	//=============================================================================
	// EXISTING DEVICES
	//=============================================================================
	#tempRetValDeviceStates := DeviceStates(LADDR := #ioSystemHwId,
	                                        MODE := #STATE_EXIST,
	                                        STATE := #statExistingDevices);

	// Check if the block call was successful
	IF (#tempRetValDeviceStates <> 0)
	THEN
	    // Error handling
	    #status := #tempRetValDeviceStates;
	    #instructionError := #ERR_DEV_STATE_DEVICES;
	    // Call ok --> store the actual number of configured devices
	ELSE
	    ;
	END_IF;

	//=============================================================================
	// FAULTY DEVICES
	//=============================================================================
	#tempRetValDeviceStates := DeviceStates(LADDR := #ioSystemHwId,
	                                        MODE := #STATE_FAULTY,
	                                        STATE := #statFaultyDevices);

	// Check if the block call was successful
	IF (#tempRetValDeviceStates <> 0)
	THEN
	    // Error handling
	    #status := #tempRetValDeviceStates;
	    #instructionError := #ERR_DEV_STATE_DEVICES;
	    // Call ok --> store the actual number of configured devices
	ELSE
	    ;
	END_IF;

	// Find out the number of the assigned IO system, to define if it is
	// a PN or DP Network
	#tempRetValGeo := LOG2GEO(LADDR := #ioSystemHwId,
	                          GEOADDR := #statGeoAddr);

	// set IO system ID
	#ioSystem.ioSystemId := #statGeoAddr.IOSYSTEM;

	// Inilize the structure for system function GEO2LOG
	#statGeoAddr.HWTYPE := #DEVICE_SLAVE;   // Hardware type 2: IO device
	// Predefine the type OF IO system. Either Profinet IO or Profibus DP
	IF ((#statGeoAddr.IOSYSTEM >= 100)
	    AND (#statGeoAddr.IOSYSTEM <= 115))
	THEN
	    #statGeoAddr.AREA := #IO_SYSTEM_AREA;   // Area ID 1: PROFINET IO
	    #statMaxDevices := #MAX_SLAVES_PN;
	ELSIF ((#statGeoAddr.IOSYSTEM >= 1)
	    AND (#statGeoAddr.IOSYSTEM <= 32))
	THEN
	    #statGeoAddr.AREA := #DP_SYSTEM_AREA;   // Area ID 1: Profibus DP
	    #statMaxDevices := #MAX_SLAVES_DP;
	ELSE
	    ;
	END_IF;

	// Go trough all devices and get the status of the configured
	FOR #tempIndex := 1 TO #statMaxDevices DO
	    // The devices are configured --> Read out the logical address and the
	    // device name
	    IF (#statConfiguredDevices[#tempIndex] = TRUE)
	    THEN
	        // Increment the actual configured devices, store the state and
	        // HW_ID as an numerical value (UINT)
	        #statActualConfiguredDevices := #statActualConfiguredDevices + 1;

	        // Store the first configured device for the linked list
	        IF (#statFirstDeviceFlag = TRUE)
	        THEN
	            #statFirstDevice := INT_TO_UINT(#tempIndex);
	            #ioSystem.firstDevice := UINT_TO_INT(#statFirstDevice);
	            #statFirstDeviceFlag := FALSE;
	            #tempLastDevice := INT_TO_UINT(#tempIndex);
	            // It is not the first bit --> Store the actual index as "next device"
	            // in the further one!
	        ELSE
	            #ioSystem.device[#tempLastDevice].nextDevice := #tempIndex;
	            #tempLastDevice := INT_TO_UINT(#tempIndex);
	        END_IF;
	        // Store the index of the last device for the exit condition of the
	        // followiing instructions
	        #statLastDevice := #tempLastDevice;
	        #ioSystem.lastDevice := UINT_TO_INT(#statLastDevice);

	        // Station number
	        #statGeoAddr.STATION := INT_TO_UINT(#tempIndex);
	        // read LADDR from devices
	        #tempRetValGeo := GEO2LOG(GEOADDR := #statGeoAddr,
	                                  LADDR => #statGeoLaddr);
	        // Everything is ok!
	        IF (#tempRetValGeo = 0)
	        THEN
	            // store LADDR from devices in diagnostic data block
	            #ioSystem.device[#tempIndex].laddr := #statGeoLaddr;

	            // Store the device name, if the device is existing
	            // Get name is an acyclic instruction. In the startup OB, the
	            // instruction has to be repeated until it is done or error
	            REPEAT
	                // Get device name of each decive in PN System
	                #instGetNameDevices(LADDR := #ioSystemHwId,
	                                    STATION_NR := #statGeoAddr.STATION,
	                                    DATA := #tempStringConvert);

	            UNTIL (#instGetNameDevices.DONE = TRUE)
	                OR (#instGetNameDevices.ERROR = TRUE)
	            END_REPEAT;

	            IF (#instGetNameDevices.ERROR = TRUE)
	            THEN
	                // Error handling
	                #status := WORD_TO_INT(#instGetNameDevices.STATUS);
	                #instructionError := #ERR_GET_NAME_DEVICES;
	                #errorIndex := #tempIndex;

	                // Everything is ok --> Convert the String[254] into String[50]
	            ELSIF (#instGetNameDevices.DONE = TRUE)
	            THEN
	                // Cut all characters more than 50 to reduce the string length
	                #ioSystem.device[#tempIndex].name := DELETE(IN := #tempStringConvert,
	                                                            L := 204,
	                                                            P := 50);

	                // Initialize the temporary string before next loop
	                #tempStringConvert := #statInitString;
	            ELSE
	                ;
	            END_IF;
	        ELSE
	            // If the return value ist not = 0 --> the device/system/module is
	            // not configured --> No error handling
	            // set LADDR from devices to 0 in diagnostic data block
	            #ioSystem.device[#tempIndex].laddr := 0;
	            #ioSystem.device[#tempIndex].name := '';
	        END_IF;

	        // Check if the configured devices are faulty or lost once through
	        // the startup!
	        IF (#statExistingDevices[#tempIndex] = TRUE)
	        THEN
	            IF (#statFaultyDevices[#tempIndex] = TRUE)
	            THEN

	                #ioSystem.device[#tempIndex].errorState := 2;
	                #ioSystem.device[#tempIndex].error := TRUE;

	                // The device is not faulty and does exist --> set state ok!
	            ELSE
	                #ioSystem.device[#tempIndex].errorState := 1;
	                #ioSystem.device[#tempIndex].error := FALSE;
	            END_IF;
	            // The connection to the device is lost at the moment
	        ELSE
	            #ioSystem.device[#tempIndex].errorState := 3;
	            #ioSystem.device[#tempIndex].error := TRUE;
	        END_IF;
	        // No device is configured
	    ELSE
	        ;
	    END_IF;

	END_FOR;
	// Store the actual configured devices in the diagnostics structure
	#ioSystem.actualConfiguredDevices := #statActualConfiguredDevices;

	// Mark parameter "Next Device" of the last device in the list
	// --> "Next Device" = negative --> Last device in the list
	#ioSystem.device[#statLastDevice].nextDevice := -1;

	// Go through the devices until the last device is reached
	// If there are gaps between the device-list, jump over and have a look on
	// the "NextDevice" parameter
	REPEAT
	    IF (#statFirstRun = TRUE)
	    THEN
	        // The index of the linked list is representing the station number.
	        #statGeoAddr.STATION := #statFirstDevice;
	        // Initialize the pointer for the first run
	        #statLinkedListPointer := UINT_TO_INT(#statFirstDevice);
	        // Reset the flag, which signalizes the first run.
	        #statFirstRun := FALSE;
	    ELSE
	        // The index of the linked list is representing the station number.
	        #statGeoAddr.STATION := INT_TO_UINT(#statLinkedListPointer);
	    END_IF;

	    //=============================================================================
	    // Get the logical address of all modules and store the actual number of
	    // modules from each device
	    //=============================================================================

	    // Inilize the structure for system function GEO2LOG
	    #statGeoAddr.HWTYPE := #MODULE_OF_DEVICE;   // Hardware type 4: Module
	    FOR #tempModuleNum := 0 TO 10 DO
	        // Slot number
	        #statGeoAddr.SLOT := INT_TO_UINT(#tempModuleNum);
	        // read LADDR from modules
	        #tempRetValGeo := GEO2LOG(GEOADDR := #statGeoAddr,
	                                  LADDR => #statGeoLaddr);
	        // check Retval
	        IF (#tempRetValGeo = 0)
	        THEN
	            // store LADDR from modules in diagnostic data block
	            #ioSystem.device[#statLinkedListPointer].slot[#tempModuleNum].slotLaddr := #statGeoLaddr;
	            #ioSystem.device[#statLinkedListPointer].actualConfiguredModules := #ioSystem.device[#statLinkedListPointer].actualConfiguredModules + 1;
	        ELSE
	            // If the return value ist not = 0 --> the device/system/module is
	            // not configured --> No error handling
	            // set LADDR from modules to 0 in diagnostic data block
	            #ioSystem.device[#statLinkedListPointer].slot[#tempModuleNum].slotLaddr := 0;
	        END_IF;
	    END_FOR;

	    //=============================================================================
	    // Check modules of faulty Devices
	    //=============================================================================

	    // Check the state of the configured devices
	    IF (#ioSystem.device[#statLinkedListPointer].errorState = 2)
	    THEN
	        // The device is reachable, but faulty because of an error in a
	        // subordinated system --> check the modules
	        #tempRetValModuleStates := ModuleStates(LADDR := #ioSystem.device[#statLinkedListPointer].laddr,
	                                                MODE := #STATE_PROBLEM,
	                                                STATE := #statDeviceModuleStates);

	        IF (#tempRetValModuleStates <> 0)
	        THEN
	            // Error hanlding
	            #status := #tempRetValModuleStates;
	            #instructionError := #ERR_MOD_STAT_DEVICES;
	            #errorIndex := UINT_TO_INT(#statFirstDevice);
	        ELSE
	            // Store the state of the different module in the diag DB
	            FOR #tempSlotIndex := 0 TO #ioSystem.device[#statFirstDevice].actualConfiguredModules DO
	                IF (#statDeviceModuleStates[#tempSlotIndex + 1] = TRUE)
	                THEN
	                    #ioSystem.device[#statLinkedListPointer].slot[#tempSlotIndex].slotErrorState := TRUE;
	                ELSE
	                    #ioSystem.device[#statLinkedListPointer].slot[#tempSlotIndex].slotErrorState := FALSE;
	                END_IF;
	            END_FOR;
	        END_IF;
	    ELSIF (#ioSystem.device[#statLinkedListPointer].errorState = 3)
	    THEN

	        FOR #tempSlotIndex := 0 TO #ioSystem.device[#statLinkedListPointer].actualConfiguredModules DO
	            IF (#ioSystem.device[#statLinkedListPointer].slot[#tempSlotIndex].slotLaddr <> 0)
	            THEN
	                #ioSystem.device[#statLinkedListPointer].slot[#tempSlotIndex].slotErrorState := TRUE;
	            END_IF;
	        END_FOR;

	    ELSE
	        ; // no faulty device --> nothing to do!
	    END_IF;

	    // Initialize the pointer for the next run
	    #statLinkedListPointer := #ioSystem.device[#statLinkedListPointer].nextDevice;
	    // If the last device is reached, reset the bit for the first run
	    //#FirstRun := TRUE;
	    // Checking the modules is done, the last device is reached
	UNTIL (#statLinkedListPointer < 0)
	END_REPEAT;
	// Reset the condition for the first run.
	#statFirstRun := TRUE;


END_FUNCTION_BLOCK

DATA_BLOCK "DiagStartupIoSystem_iDB"
{ S7_Optimized_Access := 'TRUE' }
VERSION : 0.1
NON_RETAIN
"DiagStartupIoSystem"

BEGIN

END_DATA_BLOCK

FUNCTION_BLOCK "DiagStartupPlc"
{ S7_Optimized_Access := 'TRUE' }
VERSION : 0.1
   VAR_OUTPUT
      status : Int;   // The return value of system function, where the last error occured
      instructionError : Int;   // Indicates in which system function the error occured: 1= DeviceStates PN , 2=GetName PN, 3=ModuleStates PN,  4=DeviceStates DP, 5= GetName DP. 6= ModuleStates DP
   END_VAR

   VAR_IN_OUT
      plc : "typePlc";   // The diagnostics structure for one PLC
   END_VAR

   VAR
      statGeoAddr {OriginalPartName := 'GEOADDR'; LibVersion := '1.0'; ExternalAccessible := 'False'; ExternalVisible := 'False'; ExternalWritable := 'False'} : GEOADDR;   // Slot information
      statGeoLaddr { ExternalAccessible := 'False'; ExternalVisible := 'False'; ExternalWritable := 'False'} : HW_ANY;   // GEO2LOG hardware identifier
      statActualCentralModules : USInt := 0;   // Actual number of modules in the central station (PLC)
      statPlcModuleStates : Array[0..127] of Bool;   // Storage of the status of all modules in the PLC central station --> State: Problem
   END_VAR

   VAR_TEMP
      tempModuleNum : Int;   // index module number
      tempRetValGeo : Int;   // GEO2LOG error information
      tempRetValModuleStates : Int;   // Return value system function ModuleStates
   END_VAR

   VAR CONSTANT
      MODULE_OF_PLC : USInt := 4;   // GEO2LOG structure: HW type = 4
      CPU : USInt := 0;   // GEO2LOG structure: Area = 0
      CENTRAL_SYSTEM : USInt := 0;   // GEO2LOG structure: IO System = 0
      CENTRAL_STATION : USInt;   // GEO2LOG structure: Station = 0
      HW_ID_PLC_MODULES : HW_DEVICE := 32;   // HW ID of the PLC, which is needed for getting the module states --> fix value
      STATE_PROBLEM : USInt := 5;   // Used for instruction DeviceStates, read out all devices with several problems
      ERR_MOD_STAT_CENTRAL : USInt := 3;   // Value for output instruction error, ModuleStates local modules
   END_VAR


BEGIN
	//=============================================================================
	//Author: SIEMENS, Owner: Miklos Boros
	//        email: borosmiklos@gmail.com; miklos.boros@esss.se
	//
	//Functionality: Determine hardware identifier and module states from local
	//               modules
	//
	//
	//Please Note:
	//        This block is part of the generated ESS Standard Code
	//        DON'T CHANGE THIS BLOCK MANUALY. Any changes will be overwritten in the next code generation.
	//
	//
	//Change log table:
	//Version  Date         Expert in charge      Changes applied
	//01.00.00 29.08.2017   ESS/ICS               First released version for PLCFactory
	//02.00.00 09-04-2018   ESS/ICS               Major bug fix for PN/DP devices
	//=============================================================================


	//=============================================================================
	// Determine hardware identifier from LOCAL MODULES
	//=============================================================================
	#statGeoAddr.HWTYPE := #MODULE_OF_PLC;      // Hardware type 4: module
	#statGeoAddr.AREA := #CPU;                  // Area ID 0: CPU
	#statGeoAddr.IOSYSTEM := #CENTRAL_SYSTEM;   // PROFINET IO system
	                                            // (0 = central unit in the rack)
	#statGeoAddr.STATION := #CENTRAL_STATION;   // Number of the rack
	                                            // if area identifier
	                                            //  AREA = 0 (central module).

	FOR #tempModuleNum := 1 TO 10 DO
	  // Slot number
	  #statGeoAddr.SLOT := INT_TO_UINT(#tempModuleNum);
	  // read LADDR from local modules
	  #tempRetValGeo := GEO2LOG(GEOADDR := #statGeoAddr,
	                            LADDR => #statGeoLaddr);
	  // check Retval
	  IF (#tempRetValGeo = 0)
	  THEN
	    // store LADDR from local modules in diagnostic data block
	    #plc.slot[#tempModuleNum].slotLaddr := #statGeoLaddr;
	    #statActualCentralModules := #statActualCentralModules + 1;
	  ELSE
	    // If the return value ist not = 0 --> the device/system/module is not
	    // configured --> No error handling
	    // set LADDR from local modules to 0 in diagnostic data block
	    #plc.slot[#tempModuleNum].slotLaddr := 0;
	  END_IF;
	  // Store the actual configured devices in the diagnostics DB
	  #plc.actualConfiguredCentralModules := #statActualCentralModules;
	END_FOR;


	//=============================================================================
	// Check module states from LOCAL MODULES
	//=============================================================================
	// Check if central module are available - at least one module is always
	// configured, the PLC itself
	IF (#plc.actualConfiguredCentralModules > 1)
	THEN
	  // Check the status of the local modules
	  #tempRetValModuleStates := ModuleStates(LADDR := #HW_ID_PLC_MODULES,
	                                          MODE := #STATE_PROBLEM,
	                                          STATE := #statPlcModuleStates);

	  // Check if the block call was successful
	  IF (#tempRetValModuleStates <> 0)
	  THEN
	    // Error handling
	    #status := #tempRetValModuleStates;
	    #instructionError := #ERR_MOD_STAT_CENTRAL;
	  ELSE
	    ; // Everything is ok!
	  END_IF;
	ELSE
	  ; // There are no central module configured
	END_IF;

	// The error LED of the PLC is flashing --> Set error state of the PLC
	#plc.errorState := TRUE;


	//=============================================================================
	// set module states from LOCAL MODULES
	//=============================================================================

	// If the first bit in the array is true, at least one module is faulty
	IF (#statPlcModuleStates[0] = TRUE)
	THEN
	  // Check which of the modules are faulty
	  // PLC modules array starts at index 2 for the first local module
	  FOR #tempModuleNum := 2 TO #plc.actualConfiguredCentralModules + 1 DO
	    IF (#statPlcModuleStates[#tempModuleNum] = TRUE)
	    THEN
	      #plc.slot[#tempModuleNum - 1].slotErrorState := TRUE;
	    ELSE
	      #plc.slot[#tempModuleNum - 1].slotErrorState := FALSE;
	    END_IF;
	  END_FOR;

	ELSE
	  // Everything is ok!
	  FOR #tempModuleNum := 1 TO #plc.actualConfiguredCentralModules DO
	    #plc.slot[#tempModuleNum].slotErrorState := FALSE;
	  END_FOR;

	END_IF;

END_FUNCTION_BLOCK


DATA_BLOCK "DiagStartupPlc_iDB"
{ S7_Optimized_Access := 'TRUE' }
VERSION : 0.1
NON_RETAIN
"DiagStartupPlc"

BEGIN

END_DATA_BLOCK

FUNCTION "DiagnosticError" : Void
{ S7_Optimized_Access := 'TRUE' }
VERSION : 0.1
   VAR_INPUT
      ioState : Word;   // IO state of the HW object
      laddr : HW_ANY;   // Hardware identifier
      channel : UInt;   // Channel number
      multiError : Bool;   // =true if more than one error is present
   END_VAR

   VAR_IN_OUT
      plc : "typePlc";   // The diagnostics structure for one PLC
      ioSystem : Array[1..5] of "typeIoSystem";   // The diagnostics structure for one IO System
   END_VAR

   VAR_TEMP
      tempGeoAddr {OriginalPartName := 'GEOADDR'; LibVersion := '1.0'} : GEOADDR;   // Geographical address of the disturbed Module / Device
      tempIoSystemIndex : Int;   // Index for IO System
      index : Int;   // index system
      tempRetVal : Int;   // Return value of LOG2GEO
   END_VAR

   VAR CONSTANT
      GOOD : Word := 16#0001;   // Status of the hardware object: Bit 0: Good
      AREA_CENTRAL : UInt := 0;   // Area ID for PLC
      AREA_PROFINET : UInt := 1;   // Area ID for PROFINET IO
      AREA_PROFIBUS : UInt := 2;   // Area ID for PROFIBUS DP
   END_VAR


BEGIN
	//=============================================================================
	//Author: SIEMENS, Owner: Miklos Boros
	//        email: borosmiklos@gmail.com; miklos.boros@esss.se
	//
	//Functionality: Evaluate Diagnostic interrupt OB information for PLC and
	//               devices
	//
	//
	//Please Note:
	//        This block is part of the generated ESS Standard Code
	//        DON'T CHANGE THIS BLOCK MANUALY. Any changes will be overwritten in the next code generation.
	//
	//
	//Change log table:
	//Version  Date         Expert in charge      Changes applied
	//01.00.00 29-08-2017   ESS/ICS               First released version for PLCFactory
	//02.00.00 09-04-2018   ESS/ICS               Major bug fix for PN/DP devices
	//=============================================================================


	//=============================================================================
	// determine geographic address of faulty device
	//=============================================================================
	#tempRetVal := LOG2GEO(LADDR := #laddr,
	                       GEOADDR := #tempGeoAddr);


	//=============================================================================
	// evaluate diagnosis information for devices in an IO system
	//=============================================================================
	IF (#tempGeoAddr.AREA = #AREA_PROFINET)
	    OR (#tempGeoAddr.AREA = #AREA_PROFIBUS)
	THEN

	    //=============================================================================
	    // determine index for IO system
	    //=============================================================================
	    FOR #index := 1 TO 5 DO
	        IF ("DiagnosticsData".ioSystem[#index].ioSystemId = #tempGeoAddr.IOSYSTEM)
	        THEN
	            #tempIoSystemIndex := #index;
	        END_IF;
	    END_FOR;

	    IF (#tempIoSystemIndex <= 5)
	        AND (#tempGeoAddr.STATION <= 10)
	        AND (#tempGeoAddr.SLOT <= 10)
	    THEN
	        // evaluate diagnosis information IO system
	        IF (#ioState = #GOOD)
	        THEN
	            #ioSystem[#tempIoSystemIndex].device[#tempGeoAddr.STATION].error := FALSE;
	            #ioSystem[#tempIoSystemIndex].device[#tempGeoAddr.STATION].slot[#tempGeoAddr.SLOT].slotErrorState := FALSE;

	            IF (#ioSystem[#tempIoSystemIndex].device[#tempGeoAddr.STATION].errorState = 2)
	            THEN
	                #ioSystem[#tempIoSystemIndex].device[#tempGeoAddr.STATION].errorState := 12;
	            ELSIF (#ioSystem[#tempIoSystemIndex].device[#tempGeoAddr.STATION].errorState = 3)
	            THEN
	                #ioSystem[#tempIoSystemIndex].device[#tempGeoAddr.STATION].errorState := 13;
	            ELSE
	                #ioSystem[#tempIoSystemIndex].device[#tempGeoAddr.STATION].errorState := 1;
	            END_IF;
	        ELSE
	            #ioSystem[#tempIoSystemIndex].device[#tempGeoAddr.STATION].error := TRUE;
	            #ioSystem[#tempIoSystemIndex].device[#tempGeoAddr.STATION].errorState := 2;

	            #ioSystem[#tempIoSystemIndex].device[#tempGeoAddr.STATION].slot[#tempGeoAddr.SLOT].slotErrorState := TRUE;
	        END_IF;


	    END_IF;

	    //=============================================================================
	    // evaluate diagnosis information for PLC
	    //=============================================================================
	ELSIF (#tempGeoAddr.AREA = #AREA_CENTRAL)
	THEN

	    IF (#tempGeoAddr.SLOT <= 10)
	    THEN
	        // evaluate diagnosis information PLC
	        IF (#ioState = #GOOD)
	        THEN
	            #plc.slot[#tempGeoAddr.SLOT].slotErrorState := FALSE;
	        ELSE
	            #plc.slot[#tempGeoAddr.SLOT].slotErrorState := TRUE;
	        END_IF;

	    END_IF;

	ELSE
	    ;
	END_IF;

END_FUNCTION

FUNCTION "PullOrPlugModules" : Void
{ S7_Optimized_Access := 'TRUE' }
VERSION : 0.1
   VAR_INPUT
      laddr : HW_IO;   // Hardware identifier
      eventClass : Byte;   // 16#38/39: module inserted, removed
      faultId : Byte;   // Fault identifier
   END_VAR

   VAR_IN_OUT
      plc : "typePlc";   // The diagnostics structure for one PLC
      ioSystem : Array[1..5] of "typeIoSystem";   // The diagnostics structure for one IO System
   END_VAR

   VAR_TEMP
      tempIoSystemIndex : Int;   // Index for IO System
      index : Int;   // index system
      tempGeoAddr {OriginalPartName := 'GEOADDR'; LibVersion := '1.0'} : GEOADDR;   // Geographical address of the disturbed Module / Device
      tempRetVal : Int;   // Return value of LOG2GEO
   END_VAR

   VAR CONSTANT
      AREA_CENTRAL : UInt := 0;   // Area ID for PLC
      AREA_PROFINET : UInt := 1;   // Area ID for PROFINET IO
      AREA_PROFIBUS : UInt := 2;   // Area ID for PROFIBUS DP
      MODULE_PLUGGED : Byte := 16#38;   // (Sub)module plugged
      MODULE_PULLED : Byte := 16#39;   // (Sub)module pulled or not responding
      MODULE_MATCHES : Byte := 16#54;   // IO submodule inserted and matches configured submodule
      MODULE_OK : Byte := 16#61;   // Module inserted, module type OK
   END_VAR


BEGIN
	//=============================================================================
	//Author: SIEMENS, Owner: Miklos Boros
	//        email: borosmiklos@gmail.com; miklos.boros@esss.se
	//
	//Functionality: Evaluate Pull/plug interrupt OB information for PLC and
	//               devices
	//
	//
	//Please Note:
	//        This block is part of the generated ESS Standard Code
	//        DON'T CHANGE THIS BLOCK MANUALY. Any changes will be overwritten in the next code generation.
	//
	//
	//Change log table:
	//Version  Date         Expert in charge      Changes applied
	//01.00.00 29.08.2017   ESS/ICS               First released version for PLCFactory
	//02.00.00 09-04-2018   ESS/ICS               Major bug fix for PN/DP devices
	//=============================================================================


	//=============================================================================
	// determine geographic address of faulty device
	//=============================================================================
	#tempRetVal := LOG2GEO(LADDR := #laddr,
	                       GEOADDR := #tempGeoAddr);

	//=============================================================================
	// evaluate diagnosis information for devices in an IO system
	//=============================================================================
	IF (#tempGeoAddr.AREA = #AREA_PROFINET)
	    OR (#tempGeoAddr.AREA = #AREA_PROFIBUS)
	THEN

	    //=============================================================================
	    // determine index for IO system
	    //=============================================================================
	    FOR #index := 1 TO 5 DO
	        IF (#ioSystem[#index].ioSystemId = #tempGeoAddr.IOSYSTEM)
	        THEN
	            #tempIoSystemIndex := #index;
	        END_IF;
	    END_FOR;

	    IF (#tempIoSystemIndex <= 5)
	        AND (#tempGeoAddr.STATION <= 10)
	        AND (#tempGeoAddr.SLOT <= 10)
	    THEN
	        // check modules plugged
	        IF (#eventClass = #MODULE_PLUGGED)
	        THEN
	            // reset error state only if the correct module is inserted
	            IF (#faultId = #MODULE_MATCHES)
	                OR (#faultId = #MODULE_OK)
	            THEN
	                #ioSystem[#tempIoSystemIndex].device[#tempGeoAddr.STATION].error := FALSE;
	                #ioSystem[#tempIoSystemIndex].device[#tempGeoAddr.STATION].slot[#tempGeoAddr.SLOT].slotErrorState := FALSE;

	                IF (#ioSystem[#tempIoSystemIndex].device[#tempGeoAddr.STATION].errorState = 2)
	                THEN
	                    #ioSystem[#tempIoSystemIndex].device[#tempGeoAddr.STATION].errorState := 12;
	                ELSIF (#ioSystem[#tempIoSystemIndex].device[#tempGeoAddr.STATION].errorState = 3)
	                THEN
	                    #ioSystem[#tempIoSystemIndex].device[#tempGeoAddr.STATION].errorState := 13;
	                ELSE
	                    #ioSystem[#tempIoSystemIndex].device[#tempGeoAddr.STATION].errorState := 1;
	                END_IF;
	            END_IF;

	            // check modules pulled
	        ELSIF (#eventClass = #MODULE_PULLED)
	        THEN
	            #ioSystem[#tempIoSystemIndex].device[#tempGeoAddr.STATION].error := TRUE;
	            #ioSystem[#tempIoSystemIndex].device[#tempGeoAddr.STATION].errorState := 2;

	            #ioSystem[#tempIoSystemIndex].device[#tempGeoAddr.STATION].slot[#tempGeoAddr.SLOT].slotErrorState := TRUE;

	        ELSE
	            ;
	        END_IF;


	    END_IF;

	    //=============================================================================
	    // evaluate diagnosis information for PLC
	    //=============================================================================
	ELSIF (#tempGeoAddr.AREA = #AREA_CENTRAL)
	THEN

	    IF (#tempGeoAddr.SLOT <= 10)
	    THEN
	        IF (#eventClass = #MODULE_PLUGGED)
	        THEN
	            IF (#faultId = #MODULE_MATCHES)
	                OR (#faultId = #MODULE_OK)
	            THEN
	                #plc.slot[#tempGeoAddr.SLOT].slotErrorState := FALSE;
	            END_IF;

	        ELSIF (#eventClass = #MODULE_PULLED)
	        THEN
	            #plc.slot[#tempGeoAddr.SLOT].slotErrorState := TRUE;
	        ELSE
	            ;
	        END_IF;


	    END_IF;

	ELSE
	    ;
	END_IF;

END_FUNCTION

FUNCTION "RackOrStationFaliure" : Void
{ S7_Optimized_Access := 'TRUE' }
VERSION : 0.1
   VAR_INPUT
      laddr : HW_DEVICE;   // Hardware identifier
      eventClass : Byte;   // Event class
      faultId : Byte;   // Fault identifier
   END_VAR

   VAR_IN_OUT
      plc : "typePlc";   // The diagnostics structure for one PLC
      ioSystem : Array[1..5] of "typeIoSystem";   // The diagnostics structure for one IO System
   END_VAR

   VAR_TEMP
      index : Int;   // index system
      tempSlotIndex : Int;   // Loop index
      tempIoSystemIndex : Int;   // Index for IO System
      tempGeoAddr {OriginalPartName := 'GEOADDR'; LibVersion := '1.0'} : GEOADDR;   // Geographical address of the disturbed Module / Device
      tempRetVal : Int;   // Return value of LOG2GEO
      tempRetValModuleStates : Int;   // Return value system function ModuleStates
      tempDeviceModuleStates : Array[0..127] of Bool;   // Storage of the status of all modules in the PN Devices --> State: Problem
      tempLaddr : HW_DEVICE;   // logical address of the disturbed Module / Device
   END_VAR

   VAR CONSTANT
      AREA_CENTRAL : UInt := 0;   // Area ID for PLC
      AREA_PROFINET : UInt := 1;   // Area ID for PROFINET IO
      AREA_PROFIBUS : UInt := 2;   // Area ID for PROFIBUS DP
      SLAVE_DEVICE_RET : Byte := 16#38;   // return of a DP slave / IO device
      SLAVE_DEVICE_FAIL : Byte := 16#39;   // Failure of a DP slave / IO device
      DP_SLAVE_FAIL_RET : Byte := 16#C4;   // Failure/return of a DP slave
      IO_DEVICE_FAIL_RET : Byte := 16#CB;   // Failure/return of a PROFINET IO device
      STATE_PROBLEM : USInt := 5;   // Used for instruction DeviceStates, read out all devices with several problems
   END_VAR


BEGIN
	//=============================================================================
	//Author: SIEMENS, Owner: Miklos Boros
	//        email: borosmiklos@gmail.com; miklos.boros@esss.se
	//
	//Functionality: Evaluate Rack/Station interrupt OB information for PLC and
	//               devices
	//
	//
	//Please Note:
	//        This block is part of the generated ESS Standard Code
	//        DON'T CHANGE THIS BLOCK MANUALY. Any changes will be overwritten in the next code generation.
	//
	//
	//Change log table:
	//Version  Date         Expert in charge      Changes applied
	//01.00.00 29.08.2017   ESS/ICS               First released version for PLCFactory
	//02.00.00 09-04-2018   ESS/ICS               Major bug fix for PN/DP devices
	//=============================================================================


	//=============================================================================
	// determine geographic address of faulty device
	//=============================================================================
	#tempRetVal := LOG2GEO(LADDR := #laddr,
	                       GEOADDR := #tempGeoAddr);

	//=============================================================================
	// evaluate diagnosis information for devices in an IO system
	//=============================================================================
	IF (#tempGeoAddr.AREA = #AREA_PROFINET)
	  OR (#tempGeoAddr.AREA = #AREA_PROFIBUS)
	THEN

	  //===========================================================================
	  // determine index for IO system
	  //===========================================================================
	  FOR #index := 1 TO 5 DO
	    IF (#ioSystem[#index].ioSystemId = #tempGeoAddr.IOSYSTEM)
	    THEN
	      #tempIoSystemIndex := #index;
	    END_IF;
	  END_FOR;

	  IF (#tempIoSystemIndex <= 5)
	    AND (#tempGeoAddr.STATION <= 10)
	    AND (#tempGeoAddr.SLOT <= 10)
	  THEN
	    // check DP slave or IO device return
	    IF (#eventClass = #SLAVE_DEVICE_RET)
	    THEN
	      // reset error state only if the slave or device state is OK
	      IF (#faultId = #DP_SLAVE_FAIL_RET)
	        OR (#faultId = #IO_DEVICE_FAIL_RET)
	      THEN
	        #ioSystem[#tempIoSystemIndex].device[#tempGeoAddr.STATION].error := FALSE;

	        FOR #tempSlotIndex := 0 TO #ioSystem[#tempIoSystemIndex].device[#tempGeoAddr.STATION].actualConfiguredModules DO
	          #ioSystem[#tempIoSystemIndex].device[#tempGeoAddr.STATION].slot[#tempSlotIndex].slotErrorState := FALSE;
	        END_FOR;

	        IF (#ioSystem[#tempIoSystemIndex].device[#tempGeoAddr.STATION].errorState = 2)
	        THEN
	          #ioSystem[#tempIoSystemIndex].device[#tempGeoAddr.STATION].errorState := 12;
	        ELSIF (#ioSystem[#tempIoSystemIndex].device[#tempGeoAddr.STATION].errorState = 3)
	        THEN
	          #ioSystem[#tempIoSystemIndex].device[#tempGeoAddr.STATION].errorState := 13;
	        ELSE
	          #ioSystem[#tempIoSystemIndex].device[#tempGeoAddr.STATION].errorState := 1;
	        END_IF;

	      ELSE

	        // The device is reachable, but faulty because of an error in a
	        // subordinated system --> check the modules
	        #tempRetVal := GEO2LOG(LADDR => #tempLaddr,
	                               GEOADDR := #tempGeoAddr);

	        #tempRetValModuleStates := ModuleStates(LADDR := #tempLaddr,
	                                                MODE := #STATE_PROBLEM,
	                                                STATE := #tempDeviceModuleStates);

	        IF (#tempRetValModuleStates = 0)
	        THEN
	          // Store the state of the different module in the diag DB
	          FOR #tempSlotIndex := 0 TO #ioSystem[#tempIoSystemIndex].device[#tempGeoAddr.STATION].actualConfiguredModules DO
	            IF (#tempDeviceModuleStates[#tempSlotIndex + 1] = TRUE)
	            THEN
	              #ioSystem[#tempIoSystemIndex].device[#tempGeoAddr.STATION].slot[#tempSlotIndex].slotErrorState := TRUE;
	            ELSE
	              #ioSystem[#tempIoSystemIndex].device[#tempGeoAddr.STATION].slot[#tempSlotIndex].slotErrorState := FALSE;
	            END_IF;
	          END_FOR;
	        END_IF;

	        #ioSystem[#tempIoSystemIndex].device[#tempGeoAddr.STATION].errorState := 2;

	      END_IF;

	      // check DP slave or IO device failure
	    ELSIF (#eventClass = #SLAVE_DEVICE_FAIL)
	    THEN
	      #ioSystem[#tempIoSystemIndex].device[#tempGeoAddr.STATION].error := TRUE;
	      #ioSystem[#tempIoSystemIndex].device[#tempGeoAddr.STATION].errorState := 3;

	      FOR #tempSlotIndex := 0 TO #ioSystem[#tempIoSystemIndex].device[#tempGeoAddr.STATION].actualConfiguredModules DO
	        IF #ioSystem[#tempIoSystemIndex].device[#tempGeoAddr.STATION].slot[#tempSlotIndex].slotLaddr <> 0
	        THEN
	          #ioSystem[#tempIoSystemIndex].device[#tempGeoAddr.STATION].slot[#tempSlotIndex].slotErrorState := TRUE;
	        END_IF;
	      END_FOR;

	    ELSE
	      ;
	    END_IF;


	  END_IF;

	//=============================================================================
	//evaluate diagnosis information for PLC
	//=============================================================================
	ELSIF (#tempGeoAddr.AREA = #AREA_CENTRAL)
	THEN

	  IF (#tempGeoAddr.SLOT <= 10)
	  THEN
	    // check DP slave or IO device return
	    IF (#eventClass = #SLAVE_DEVICE_RET)
	    THEN
	      IF (#faultId = #DP_SLAVE_FAIL_RET)
	        OR (#faultId = #IO_DEVICE_FAIL_RET)
	      THEN
	        #plc.slot[#tempGeoAddr.SLOT].slotErrorState := FALSE;
	      END_IF;

	      // check DP slave or IO device failure
	    ELSIF (#eventClass = #SLAVE_DEVICE_FAIL)
	    THEN
	      #plc.slot[#tempGeoAddr.SLOT].slotErrorState := TRUE;
	    ELSE
	      ;
	    END_IF;


	  END_IF;

	ELSE
	  ;
	END_IF;

END_FUNCTION

FUNCTION_BLOCK "Diagnostics"
{ S7_Optimized_Access := 'TRUE' }
VERSION : 0.1
   VAR_IN_OUT
      plc : "typePlc";   // The diagnostics structure for one PLC
      ioSystem : Array[1..5] of "typeIoSystem";   // The diagnostics structure for one IO System
   END_VAR

   VAR
      statIoSystemIndex : Int;   // Index for IO System
      statSlotIndex : Int;   // Index for Slot
      statDeviceIndex : Int;   // Index for Device
   END_VAR

   VAR_TEMP
      retValLed : Int;
   END_VAR

   VAR CONSTANT
      ERROR_LED : UInt := 2;   // Identification number of the ERROR LED
      ERROR_LED_ON : UInt := 4;   // LED status Color 1 flashing
   END_VAR


BEGIN
	//=============================================================================
	//Author: SIEMENS, Owner: Miklos Boros
	//        email: borosmiklos@gmail.com; miklos.boros@esss.se
	//
	//Functionality: Basic diagnostic function that has to be called in every cycle
	//
	//
	//Please Note:
	//        This block is part of the generated ESS Standard Code
	//        DON'T CHANGE THIS BLOCK MANUALY. Any changes will be overwritten in the next code generation.
	//
	//
	//Change log table:
	//Version  Date         Expert in charge      Changes applied
	//01.00.00 29.08.2017   ESS/ICS               First released version for PLCFactory
	//02.00.00 09-04-2018   ESS/ICS               Major bug fix for PN/DP devices
	//=============================================================================


	//=============================================================================
	// check error active
	//=============================================================================
	#retValLed := LED(LADDR := "Local~Common", LED := #ERROR_LED);
	IF #retValLed = #ERROR_LED_ON
	THEN
	    #plc.errorState := TRUE;
	ELSE
	    #plc.errorState := FALSE;
	END_IF;

	//=============================================================================
	// check error in IO systems active
	//=============================================================================
	FOR #statIoSystemIndex := 1 TO 5 DO
	    #ioSystem[#statIoSystemIndex].ioSystemError := FALSE;

	    FOR #statDeviceIndex := 1 TO 1 DO
	        IF (#ioSystem[#statIoSystemIndex].device[#statDeviceIndex].error = TRUE)
	        THEN
	            #ioSystem[#statIoSystemIndex].ioSystemError := TRUE;
	        END_IF;
	    END_FOR;
	END_FOR;



END_FUNCTION_BLOCK

DATA_BLOCK "Diagnostics_iDB"
{ S7_Optimized_Access := 'TRUE' }
VERSION : 0.1
NON_RETAIN
"Diagnostics"

BEGIN

END_DATA_BLOCK

ORGANIZATION_BLOCK "CyclicDiagnostics"
TITLE = "Main Program Sweep (Cycle)"
{ S7_Optimized_Access := 'TRUE' }
VERSION : 0.1

BEGIN
	//=============================================================================
	//Author: SIEMENS, Owner: Miklos Boros
	//        email: borosmiklos@gmail.com; miklos.boros@esss.se
	//
	//Functionality: Main Cycle OB for diagnostics
	//               OB type: Program cycle
	//
	//
	//Please Note:
	//        This block is part of the generated ESS Standard Code
	//        DON'T CHANGE THIS BLOCK MANUALY. Any changes will be overwritten in the next code generation.
	//
	//
	//Change log table:
	//Version  Date         Expert in charge      Changes applied
	//01.00.00 29-08-2017   ESS/ICS               First released version for PLCFactory
	//02.00.00 09-04-2018   ESS/ICS               Major bug fix for PN/DP devices
	//=============================================================================



	"Diagnostics_iDB"(plc:="DiagnosticsData".plc,
	                  ioSystem:="DiagnosticsData".ioSystem);

END_ORGANIZATION_BLOCK


ORGANIZATION_BLOCK "Diagnostic error interrupt"
{ S7_Optimized_Access := 'TRUE' }
VERSION : 0.1

BEGIN
	//=============================================================================
	//Author: SIEMENS, Owner: Miklos Boros
	//        email: borosmiklos@gmail.com; miklos.boros@esss.se
	//
	//Functionality: Diagnostics Error Interrupt OB
	//               OB type: Diagnostic Interrupt
	//
	//
	//Please Note:
	//        This block is part of the generated ESS Standard Code
	//        DON'T CHANGE THIS BLOCK MANUALY. Any changes will be overwritten in the next code generation.
	//
	//
	//Change log table:
	//Version  Date         Expert in charge      Changes applied
	//01.00.00 29-08-2017   ESS/ICS               First released version for PLCFactory
	//02.00.00 09-04-2018   ESS/ICS               Major bug fix for PN/DP devices
	//=============================================================================

	//
	"DiagnosticError"(ioState:=#IO_State,
	                  laddr:=#LADDR,
	                  channel:=#Channel,
	                  multiError:=#MultiError,
	                  plc:="DiagnosticsData".plc,
	                  ioSystem:="DiagnosticsData".ioSystem);

END_ORGANIZATION_BLOCK

ORGANIZATION_BLOCK "Pull or plug of modules"
{ S7_Optimized_Access := 'TRUE' }
VERSION : 0.1

BEGIN
	//=============================================================================
	//Author: SIEMENS, Owner: Miklos Boros
	//        email: borosmiklos@gmail.com; miklos.boros@esss.se
	//
	//Functionality: Pull or Plug of mudules OB
	//               OB type: Pull or Plug of devices
	//
	//
	//Please Note:
	//        This block is part of the generated ESS Standard Code
	//        DON'T CHANGE THIS BLOCK MANUALY. Any changes will be overwritten in the next code generation.
	//
	//
	//Change log table:
	//Version  Date         Expert in charge      Changes applied
	//01.00.00 29-08-2017   ESS/ICS               First released version for PLCFactory
	//02.00.00 09-04-2018   ESS/ICS               Major bug fix for PN/DP devices
	//=============================================================================

	"PullOrPlugModules"(laddr:=#LADDR,
	                    eventClass:=#Event_Class,
	                    faultId:=#Fault_ID,
	                    plc:="DiagnosticsData".plc,
	                    ioSystem:="DiagnosticsData".ioSystem);

END_ORGANIZATION_BLOCK

ORGANIZATION_BLOCK "Rack or station failure"
{ S7_Optimized_Access := 'TRUE' }
VERSION : 0.1

BEGIN
	//=============================================================================
	//Author: SIEMENS, Owner: Miklos Boros
	//        email: borosmiklos@gmail.com; miklos.boros@esss.se
	//
	//Functionality: Rack or Station faliure OB
	//               OB type: Rack or station failure
	//
	//
	//Please Note:
	//        This block is part of the generated ESS Standard Code
	//        DON'T CHANGE THIS BLOCK MANUALY. Any changes will be overwritten in the next code generation.
	//
	//
	//Change log table:
	//Version  Date         Expert in charge      Changes applied
	//01.00.00 29-08-2017   ESS/ICS               First released version for PLCFactory
	//02.00.00 09-04-2018   ESS/ICS               Major bug fix for PN/DP devices
	//=============================================================================

	"RackOrStationFaliure"(laddr:=#LADDR,
	                       eventClass:=#Event_Class,
	                       faultId:=#Fault_ID,
	                       plc:="DiagnosticsData".plc,
	                       ioSystem:="DiagnosticsData".ioSystem);

END_ORGANIZATION_BLOCK

ORGANIZATION_BLOCK "Startup"
TITLE = "Complete Restart"
{ S7_Optimized_Access := 'TRUE' }
VERSION : 0.1

BEGIN
	//=============================================================================
	//Author: SIEMENS, Owner: Miklos Boros
	//        email: borosmiklos@gmail.com; miklos.boros@esss.se
	//
	//Functionality:
	//        This OB is a Startup OB, it will be called after OB100 and before the main cycle.
	//
	//
	//Please Note:
	//        This block is part of the generated ESS Standard Code however you should use
	//        the proper ioSystem ID from the
	//
	//Change log table:
	//Version  Date         Expert in charge      Changes applied
	//01.00.00 29.08.2017   ESS/ICS               First released version for PLCFactory
	//02.00.00 09-04-2018   ESS/ICS               Major bug fix for PN/DP devices
	//=============================================================================

	//Initialize the Main PLC Diagnostic
	"DiagStartupPlc_iDB"(plc:="DiagnosticsData".plc);


	//Put your current IO device configuration here. HW identifiers are in the PLC Tags/System constants!
	//Initialize IOSystem1
	//"DiagStartupIoSystem_iDB"(ioSystemHwId:=268,
	//                          ioSystem:="DiagnosticsData".ioSystem[1]);




END_ORGANIZATION_BLOCK

FUNCTION "_CommsEPICSDataMap" : Void
{ S7_Optimized_Access := 'FALSE' }
VERSION : 0.1
   VAR_TEMP
       tHashDint : DInt;
       wordTOdint AT tHashDint : Array[0..1] of Word;
       PLC_Hash : DInt;
       IOC_Hash : DInt;
   END_VAR

   BEGIN

   // PLC Hash (Generated from PLC Factory)
   #PLC_Hash := DINT#733470530;

   // Send the PLC Hash to the EPICS IOC
   "PLCToEPICS"."Word"[1] := DINT_TO_WORD(#PLC_Hash);
   "PLCToEPICS"."Word"[0] := DINT_TO_WORD(SHR(IN := #PLC_Hash, N := 16));

   // Get Hash from the EPICS IOC
   #wordTOdint[0] := "EPICSToPLC"."Word"[0];
   #wordTOdint[1] := "EPICSToPLC"."Word"[1];
   #IOC_Hash := #tHashDint;

   // Hashes Comparison
   IF (#PLC_Hash = #IOC_Hash) THEN

      // KG-GTA:ODH-PLC-01: PLC <-> EPICS Communication Mapping
      //------------------------------------------------------------------------

      "_CommsEPICSDataMappingFBFactory"(EPICSToPLCLength           := 0,
                                        EPICSToPLCDataBlockOffset  := 10,
                                        EPICSToPLCParametersStart  := 0,
                                        PLCToEPICSLength           := 1,
                                        PLCToEPICSDataBlockOffset  := 10,
                                        EPICSToPLCCommandRegisters := "DEV_CTLG-CS:ODH-Area_iDB".CommandReg,
                                        PLCToEPICSStatusRegisters  := "DEV_CTLG-CS:ODH-Area_iDB".StatusReg,
                                        EPICSToPLCDataBlock        := "EPICSToPLC"."Word",
                                        PLCToEPICSDataBlock        := "PLCToEPICS"."Word");

      "_CommsEPICSDataMappingFBFactory"(EPICSToPLCLength           := 0,
                                        EPICSToPLCDataBlockOffset  := 10,
                                        EPICSToPLCParametersStart  := 0,
                                        PLCToEPICSLength           := 1,
                                        PLCToEPICSDataBlockOffset  := 11,
                                        EPICSToPLCCommandRegisters := "DEV_CXB-CXH:ODH-Area_iDB".CommandReg,
                                        PLCToEPICSStatusRegisters  := "DEV_CXB-CXH:ODH-Area_iDB".StatusReg,
                                        EPICSToPLCDataBlock        := "EPICSToPLC"."Word",
                                        PLCToEPICSDataBlock        := "PLCToEPICS"."Word");

      "_CommsEPICSDataMappingFBFactory"(EPICSToPLCLength           := 0,
                                        EPICSToPLCDataBlockOffset  := 10,
                                        EPICSToPLCParametersStart  := 0,
                                        PLCToEPICSLength           := 3,
                                        PLCToEPICSDataBlockOffset  := 12,
                                        EPICSToPLCCommandRegisters := "DEV_CTLG-CS:ODH-O2iM-20_iDB".CommandReg,
                                        PLCToEPICSStatusRegisters  := "DEV_CTLG-CS:ODH-O2iM-20_iDB".StatusReg,
                                        EPICSToPLCDataBlock        := "EPICSToPLC"."Word",
                                        PLCToEPICSDataBlock        := "PLCToEPICS"."Word");

      "_CommsEPICSDataMappingFBFactory"(EPICSToPLCLength           := 0,
                                        EPICSToPLCDataBlockOffset  := 10,
                                        EPICSToPLCParametersStart  := 0,
                                        PLCToEPICSLength           := 3,
                                        PLCToEPICSDataBlockOffset  := 15,
                                        EPICSToPLCCommandRegisters := "DEV_CTLG-CS:ODH-O2iM-21_iDB".CommandReg,
                                        PLCToEPICSStatusRegisters  := "DEV_CTLG-CS:ODH-O2iM-21_iDB".StatusReg,
                                        EPICSToPLCDataBlock        := "EPICSToPLC"."Word",
                                        PLCToEPICSDataBlock        := "PLCToEPICS"."Word");

      "_CommsEPICSDataMappingFBFactory"(EPICSToPLCLength           := 0,
                                        EPICSToPLCDataBlockOffset  := 10,
                                        EPICSToPLCParametersStart  := 0,
                                        PLCToEPICSLength           := 3,
                                        PLCToEPICSDataBlockOffset  := 18,
                                        EPICSToPLCCommandRegisters := "DEV_CTLG-CS:ODH-O2iM-22_iDB".CommandReg,
                                        PLCToEPICSStatusRegisters  := "DEV_CTLG-CS:ODH-O2iM-22_iDB".StatusReg,
                                        EPICSToPLCDataBlock        := "EPICSToPLC"."Word",
                                        PLCToEPICSDataBlock        := "PLCToEPICS"."Word");

      "_CommsEPICSDataMappingFBFactory"(EPICSToPLCLength           := 0,
                                        EPICSToPLCDataBlockOffset  := 10,
                                        EPICSToPLCParametersStart  := 0,
                                        PLCToEPICSLength           := 3,
                                        PLCToEPICSDataBlockOffset  := 21,
                                        EPICSToPLCCommandRegisters := "DEV_CXB-CXH:ODH-O2iM-13_iDB".CommandReg,
                                        PLCToEPICSStatusRegisters  := "DEV_CXB-CXH:ODH-O2iM-13_iDB".StatusReg,
                                        EPICSToPLCDataBlock        := "EPICSToPLC"."Word",
                                        PLCToEPICSDataBlock        := "PLCToEPICS"."Word");

      "_CommsEPICSDataMappingFBFactory"(EPICSToPLCLength           := 0,
                                        EPICSToPLCDataBlockOffset  := 10,
                                        EPICSToPLCParametersStart  := 0,
                                        PLCToEPICSLength           := 3,
                                        PLCToEPICSDataBlockOffset  := 24,
                                        EPICSToPLCCommandRegisters := "DEV_CXB-CXH:ODH-O2iM-14_iDB".CommandReg,
                                        PLCToEPICSStatusRegisters  := "DEV_CXB-CXH:ODH-O2iM-14_iDB".StatusReg,
                                        EPICSToPLCDataBlock        := "EPICSToPLC"."Word",
                                        PLCToEPICSDataBlock        := "PLCToEPICS"."Word");

      "_CommsEPICSDataMappingFBFactory"(EPICSToPLCLength           := 0,
                                        EPICSToPLCDataBlockOffset  := 10,
                                        EPICSToPLCParametersStart  := 0,
                                        PLCToEPICSLength           := 3,
                                        PLCToEPICSDataBlockOffset  := 27,
                                        EPICSToPLCCommandRegisters := "DEV_CXB-CXH:ODH-O2iM-15_iDB".CommandReg,
                                        PLCToEPICSStatusRegisters  := "DEV_CXB-CXH:ODH-O2iM-15_iDB".StatusReg,
                                        EPICSToPLCDataBlock        := "EPICSToPLC"."Word",
                                        PLCToEPICSDataBlock        := "PLCToEPICS"."Word");

      "_CommsEPICSDataMappingFBFactory"(EPICSToPLCLength           := 0,
                                        EPICSToPLCDataBlockOffset  := 10,
                                        EPICSToPLCParametersStart  := 0,
                                        PLCToEPICSLength           := 3,
                                        PLCToEPICSDataBlockOffset  := 30,
                                        EPICSToPLCCommandRegisters := "DEV_CXB-CXH:ODH-O2iM-16_iDB".CommandReg,
                                        PLCToEPICSStatusRegisters  := "DEV_CXB-CXH:ODH-O2iM-16_iDB".StatusReg,
                                        EPICSToPLCDataBlock        := "EPICSToPLC"."Word",
                                        PLCToEPICSDataBlock        := "PLCToEPICS"."Word");

      "_CommsEPICSDataMappingFBFactory"(EPICSToPLCLength           := 0,
                                        EPICSToPLCDataBlockOffset  := 10,
                                        EPICSToPLCParametersStart  := 0,
                                        PLCToEPICSLength           := 3,
                                        PLCToEPICSDataBlockOffset  := 33,
                                        EPICSToPLCCommandRegisters := "DEV_CXB-CXH:ODH-O2iM-17_iDB".CommandReg,
                                        PLCToEPICSStatusRegisters  := "DEV_CXB-CXH:ODH-O2iM-17_iDB".StatusReg,
                                        EPICSToPLCDataBlock        := "EPICSToPLC"."Word",
                                        PLCToEPICSDataBlock        := "PLCToEPICS"."Word");

      "_CommsEPICSDataMappingFBFactory"(EPICSToPLCLength           := 0,
                                        EPICSToPLCDataBlockOffset  := 10,
                                        EPICSToPLCParametersStart  := 0,
                                        PLCToEPICSLength           := 3,
                                        PLCToEPICSDataBlockOffset  := 36,
                                        EPICSToPLCCommandRegisters := "DEV_CXB-CXH:ODH-O2iM-18_iDB".CommandReg,
                                        PLCToEPICSStatusRegisters  := "DEV_CXB-CXH:ODH-O2iM-18_iDB".StatusReg,
                                        EPICSToPLCDataBlock        := "EPICSToPLC"."Word",
                                        PLCToEPICSDataBlock        := "PLCToEPICS"."Word");

      "_CommsEPICSDataMappingFBFactory"(EPICSToPLCLength           := 0,
                                        EPICSToPLCDataBlockOffset  := 10,
                                        EPICSToPLCParametersStart  := 0,
                                        PLCToEPICSLength           := 3,
                                        PLCToEPICSDataBlockOffset  := 39,
                                        EPICSToPLCCommandRegisters := "DEV_CXB-CXH:ODH-O2iM-19_iDB".CommandReg,
                                        PLCToEPICSStatusRegisters  := "DEV_CXB-CXH:ODH-O2iM-19_iDB".StatusReg,
                                        EPICSToPLCDataBlock        := "EPICSToPLC"."Word",
                                        PLCToEPICSDataBlock        := "PLCToEPICS"."Word");

      "_CommsEPICSDataMappingFBFactory"(EPICSToPLCLength           := 0,
                                        EPICSToPLCDataBlockOffset  := 10,
                                        EPICSToPLCParametersStart  := 0,
                                        PLCToEPICSLength           := 3,
                                        PLCToEPICSDataBlockOffset  := 42,
                                        EPICSToPLCCommandRegisters := "DEV_HCB-ACH:ODH-O2iM-1_iDB".CommandReg,
                                        PLCToEPICSStatusRegisters  := "DEV_HCB-ACH:ODH-O2iM-1_iDB".StatusReg,
                                        EPICSToPLCDataBlock        := "EPICSToPLC"."Word",
                                        PLCToEPICSDataBlock        := "PLCToEPICS"."Word");

      "_CommsEPICSDataMappingFBFactory"(EPICSToPLCLength           := 0,
                                        EPICSToPLCDataBlockOffset  := 10,
                                        EPICSToPLCParametersStart  := 0,
                                        PLCToEPICSLength           := 3,
                                        PLCToEPICSDataBlockOffset  := 45,
                                        EPICSToPLCCommandRegisters := "DEV_HCB-ACH:ODH-O2iM-2_iDB".CommandReg,
                                        PLCToEPICSStatusRegisters  := "DEV_HCB-ACH:ODH-O2iM-2_iDB".StatusReg,
                                        EPICSToPLCDataBlock        := "EPICSToPLC"."Word",
                                        PLCToEPICSDataBlock        := "PLCToEPICS"."Word");

      "_CommsEPICSDataMappingFBFactory"(EPICSToPLCLength           := 0,
                                        EPICSToPLCDataBlockOffset  := 10,
                                        EPICSToPLCParametersStart  := 0,
                                        PLCToEPICSLength           := 3,
                                        PLCToEPICSDataBlockOffset  := 48,
                                        EPICSToPLCCommandRegisters := "DEV_HCB-ACH:ODH-O2iM-3_iDB".CommandReg,
                                        PLCToEPICSStatusRegisters  := "DEV_HCB-ACH:ODH-O2iM-3_iDB".StatusReg,
                                        EPICSToPLCDataBlock        := "EPICSToPLC"."Word",
                                        PLCToEPICSDataBlock        := "PLCToEPICS"."Word");

      "_CommsEPICSDataMappingFBFactory"(EPICSToPLCLength           := 0,
                                        EPICSToPLCDataBlockOffset  := 10,
                                        EPICSToPLCParametersStart  := 0,
                                        PLCToEPICSLength           := 3,
                                        PLCToEPICSDataBlockOffset  := 51,
                                        EPICSToPLCCommandRegisters := "DEV_HCB-ACH:ODH-O2iM-4_iDB".CommandReg,
                                        PLCToEPICSStatusRegisters  := "DEV_HCB-ACH:ODH-O2iM-4_iDB".StatusReg,
                                        EPICSToPLCDataBlock        := "EPICSToPLC"."Word",
                                        PLCToEPICSDataBlock        := "PLCToEPICS"."Word");

      "_CommsEPICSDataMappingFBFactory"(EPICSToPLCLength           := 0,
                                        EPICSToPLCDataBlockOffset  := 10,
                                        EPICSToPLCParametersStart  := 0,
                                        PLCToEPICSLength           := 3,
                                        PLCToEPICSDataBlockOffset  := 54,
                                        EPICSToPLCCommandRegisters := "DEV_HCB-ACH:ODH-O2iM-5_iDB".CommandReg,
                                        PLCToEPICSStatusRegisters  := "DEV_HCB-ACH:ODH-O2iM-5_iDB".StatusReg,
                                        EPICSToPLCDataBlock        := "EPICSToPLC"."Word",
                                        PLCToEPICSDataBlock        := "PLCToEPICS"."Word");

      "_CommsEPICSDataMappingFBFactory"(EPICSToPLCLength           := 0,
                                        EPICSToPLCDataBlockOffset  := 10,
                                        EPICSToPLCParametersStart  := 0,
                                        PLCToEPICSLength           := 3,
                                        PLCToEPICSDataBlockOffset  := 57,
                                        EPICSToPLCCommandRegisters := "DEV_HCB-DogSh:ODH-O2iM-12_iDB".CommandReg,
                                        PLCToEPICSStatusRegisters  := "DEV_HCB-DogSh:ODH-O2iM-12_iDB".StatusReg,
                                        EPICSToPLCDataBlock        := "EPICSToPLC"."Word",
                                        PLCToEPICSDataBlock        := "PLCToEPICS"."Word");

      "_CommsEPICSDataMappingFBFactory"(EPICSToPLCLength           := 0,
                                        EPICSToPLCDataBlockOffset  := 10,
                                        EPICSToPLCParametersStart  := 0,
                                        PLCToEPICSLength           := 3,
                                        PLCToEPICSDataBlockOffset  := 60,
                                        EPICSToPLCCommandRegisters := "DEV_HCB-HPGS:ODH-O2iM-10_iDB".CommandReg,
                                        PLCToEPICSStatusRegisters  := "DEV_HCB-HPGS:ODH-O2iM-10_iDB".StatusReg,
                                        EPICSToPLCDataBlock        := "EPICSToPLC"."Word",
                                        PLCToEPICSDataBlock        := "PLCToEPICS"."Word");

      "_CommsEPICSDataMappingFBFactory"(EPICSToPLCLength           := 0,
                                        EPICSToPLCDataBlockOffset  := 10,
                                        EPICSToPLCParametersStart  := 0,
                                        PLCToEPICSLength           := 3,
                                        PLCToEPICSDataBlockOffset  := 63,
                                        EPICSToPLCCommandRegisters := "DEV_HCB-HPGS:ODH-O2iM-11_iDB".CommandReg,
                                        PLCToEPICSStatusRegisters  := "DEV_HCB-HPGS:ODH-O2iM-11_iDB".StatusReg,
                                        EPICSToPLCDataBlock        := "EPICSToPLC"."Word",
                                        PLCToEPICSDataBlock        := "PLCToEPICS"."Word");

      "_CommsEPICSDataMappingFBFactory"(EPICSToPLCLength           := 0,
                                        EPICSToPLCDataBlockOffset  := 10,
                                        EPICSToPLCParametersStart  := 0,
                                        PLCToEPICSLength           := 3,
                                        PLCToEPICSDataBlockOffset  := 66,
                                        EPICSToPLCCommandRegisters := "DEV_HCB-TCH:ODH-O2iM-6_iDB".CommandReg,
                                        PLCToEPICSStatusRegisters  := "DEV_HCB-TCH:ODH-O2iM-6_iDB".StatusReg,
                                        EPICSToPLCDataBlock        := "EPICSToPLC"."Word",
                                        PLCToEPICSDataBlock        := "PLCToEPICS"."Word");

      "_CommsEPICSDataMappingFBFactory"(EPICSToPLCLength           := 0,
                                        EPICSToPLCDataBlockOffset  := 10,
                                        EPICSToPLCParametersStart  := 0,
                                        PLCToEPICSLength           := 3,
                                        PLCToEPICSDataBlockOffset  := 69,
                                        EPICSToPLCCommandRegisters := "DEV_HCB-TCH:ODH-O2iM-7_iDB".CommandReg,
                                        PLCToEPICSStatusRegisters  := "DEV_HCB-TCH:ODH-O2iM-7_iDB".StatusReg,
                                        EPICSToPLCDataBlock        := "EPICSToPLC"."Word",
                                        PLCToEPICSDataBlock        := "PLCToEPICS"."Word");

      "_CommsEPICSDataMappingFBFactory"(EPICSToPLCLength           := 0,
                                        EPICSToPLCDataBlockOffset  := 10,
                                        EPICSToPLCParametersStart  := 0,
                                        PLCToEPICSLength           := 3,
                                        PLCToEPICSDataBlockOffset  := 72,
                                        EPICSToPLCCommandRegisters := "DEV_HCB-TCH:ODH-O2iM-8_iDB".CommandReg,
                                        PLCToEPICSStatusRegisters  := "DEV_HCB-TCH:ODH-O2iM-8_iDB".StatusReg,
                                        EPICSToPLCDataBlock        := "EPICSToPLC"."Word",
                                        PLCToEPICSDataBlock        := "PLCToEPICS"."Word");

      "_CommsEPICSDataMappingFBFactory"(EPICSToPLCLength           := 0,
                                        EPICSToPLCDataBlockOffset  := 10,
                                        EPICSToPLCParametersStart  := 0,
                                        PLCToEPICSLength           := 3,
                                        PLCToEPICSDataBlockOffset  := 75,
                                        EPICSToPLCCommandRegisters := "DEV_HCB-TCH:ODH-O2iM-9_iDB".CommandReg,
                                        PLCToEPICSStatusRegisters  := "DEV_HCB-TCH:ODH-O2iM-9_iDB".StatusReg,
                                        EPICSToPLCDataBlock        := "EPICSToPLC"."Word",
                                        PLCToEPICSDataBlock        := "PLCToEPICS"."Word");

      "_CommsEPICSDataMappingFBFactory"(EPICSToPLCLength           := 0,
                                        EPICSToPLCDataBlockOffset  := 10,
                                        EPICSToPLCParametersStart  := 0,
                                        PLCToEPICSLength           := 1,
                                        PLCToEPICSDataBlockOffset  := 78,
                                        EPICSToPLCCommandRegisters := "DEV_CXB-CXH:ODH-RIO-2_iDB".CommandReg,
                                        PLCToEPICSStatusRegisters  := "DEV_CXB-CXH:ODH-RIO-2_iDB".StatusReg,
                                        EPICSToPLCDataBlock        := "EPICSToPLC"."Word",
                                        PLCToEPICSDataBlock        := "PLCToEPICS"."Word");

      "_CommsEPICSDataMappingFBFactory"(EPICSToPLCLength           := 0,
                                        EPICSToPLCDataBlockOffset  := 10,
                                        EPICSToPLCParametersStart  := 0,
                                        PLCToEPICSLength           := 1,
                                        PLCToEPICSDataBlockOffset  := 79,
                                        EPICSToPLCCommandRegisters := "DEV_HCB-ACH:ODH-RIO-1_iDB".CommandReg,
                                        PLCToEPICSStatusRegisters  := "DEV_HCB-ACH:ODH-RIO-1_iDB".StatusReg,
                                        EPICSToPLCDataBlock        := "EPICSToPLC"."Word",
                                        PLCToEPICSDataBlock        := "PLCToEPICS"."Word");

      "_CommsEPICSDataMappingFBFactory"(EPICSToPLCLength           := 0,
                                        EPICSToPLCDataBlockOffset  := 10,
                                        EPICSToPLCParametersStart  := 0,
                                        PLCToEPICSLength           := 1,
                                        PLCToEPICSDataBlockOffset  := 80,
                                        EPICSToPLCCommandRegisters := "DEV_TS2-020Row:CnPw-U-001_iDB".CommandReg,
                                        PLCToEPICSStatusRegisters  := "DEV_TS2-020Row:CnPw-U-001_iDB".StatusReg,
                                        EPICSToPLCDataBlock        := "EPICSToPLC"."Word",
                                        PLCToEPICSDataBlock        := "PLCToEPICS"."Word");


   END_IF;

END_FUNCTION

//########## EPICS->PLC datablock ##########
DATA_BLOCK "EPICSToPLC"
{ S7_Optimized_Access := 'FALSE' }
VERSION : 0.1
   STRUCT
      "Word" : Array[0..9] of Word;
   END_STRUCT;


BEGIN
END_DATA_BLOCK

//########## PLC->EPICS datablock ##########
DATA_BLOCK "PLCToEPICS"
{ S7_Optimized_Access := 'FALSE' }
VERSION : 0.1
NON_RETAIN
   STRUCT
      "Word" : Array[0..80] of Word;
   END_STRUCT;


BEGIN
END_DATA_BLOCK

FUNCTION "_CommsEPICS" : Void
{ S7_Optimized_Access := 'TRUE' }
VERSION : 0.1

BEGIN
	//Heartbeat PLC->EPICS
	IF "Utilities".Pulse_1s THEN
	    "PLCToEPICS"."Word"[2] := "PLCToEPICS"."Word"[2] + 1;
	    IF "PLCToEPICS"."Word"[2] >= 32000 THEN
	        "PLCToEPICS"."Word"[2] := 0;
	    END_IF;
	END_IF;

	// Call the comms block to provide PLC<->EPICS comms
	"_CommsPLC_EPICS_DB"(Enable         := "Utilities".AlwaysOn,
	                     SendTrigger    := "Utilities".Pulse_200ms,
	                     BytesToSend    := 162,
	                     InterfaceID    := 64,
	                     S7ConnectionID := 256,
	                     MBConnectionID := 255,
	                     S7Port         := 2000,
	                     MBPort         := 502,
	                     PLCToEPICSData := "PLCToEPICS"."Word",
	                     EPICSToPLCData := "EPICSToPLC"."Word");

	//Map all devices command and status registers to EPICS->PLC and PLC->EPICS data exchange blocks
	"_CommsEPICSDataMap"();

END_FUNCTION

